// TIA Portal V17 export
// export: Created 2021-12-03T08:13:11.4978392Z, ExportSetting WithDefaults, DisplayName Totally Integrated Automation Portal, DisplayVersion V17, DisplayName TIA Portal Openness, DisplayVersion V17, DisplayName TIA Portal Version Control Interface, DisplayVersion V17, DisplayName STEP 7 Professional, DisplayVersion V17, DisplayName STEP 7 Safety, DisplayVersion V17, DisplayName WinCC Advanced, DisplayVersion V17
FUNCTION_BLOCK "FFB_TmSel"   // FB700, F_FBD
VERSION : 0.1
// stored: AutoNumber false, IsIECCheckEnabled false, UDAEnableTagReadback false
   VAR_INPUT
      I_Sel_2 : Bool;   // Selector (0=Time 1 / 1=Time 2)
      I_Time_1 : Time;   // Time 1
      I_Time_2 : Time;   // Time 2
   END_VAR
   VAR_OUTPUT
      O_Sel_2 : Bool;
      O_SelTime : Time;   // Selected Time
   END_VAR
BEGIN

REGION Network 1
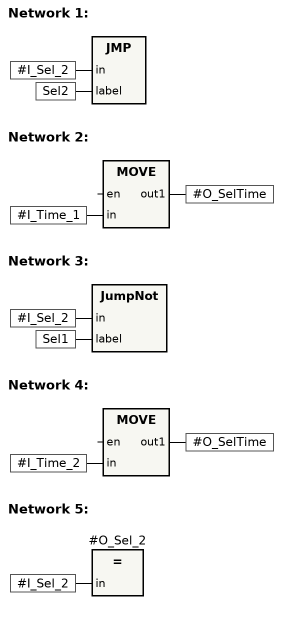
   IF #I_Sel_2 THEN GOTO Sel2; END_IF;
END_REGION

REGION Network 2
   #O_SelTime := #I_Time_1;
END_REGION

REGION Network 3
   // no SCL statement known for JumpNot: written as a call
   JumpNot(in := #I_Sel_2, label := Sel1);
END_REGION

REGION Network 4
   Sel2:
   #O_SelTime := #I_Time_2;
END_REGION

REGION Network 5
   Sel1:
   #O_Sel_2 := #I_Sel_2;
END_REGION
END_FUNCTION_BLOCK
